PROGRAM Jog_Axis
VAR
	fbJog: MC_Jog;
	JogForwardPB: BOOL;
	JogBackwardsPB: BOOL;
END_VAR

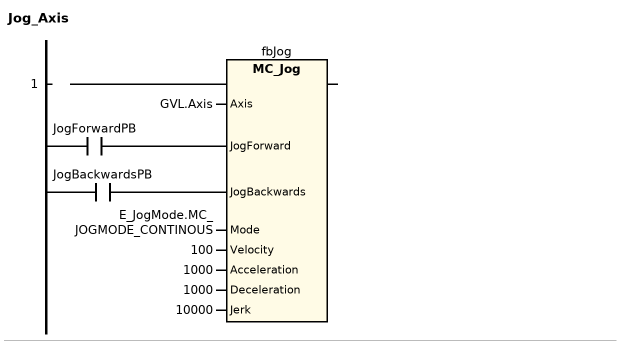
// NETWORK 1
fbJog(
    Axis := GVL.Axis,
    JogForward := JogForwardPB,
    JogBackwards := JogBackwardsPB,
    Mode := E_JogMode.MC_JOGMODE_CONTINOUS,
    Velocity := 100,
    Acceleration := 1000,
    Deceleration := 1000,
    Jerk := 10000); // MC_Jog

END_PROGRAM

(* stored: Version 1.1.0.1, ProductVersion 3.1.4024.12
   POU Jog_Axis: Id {cc0138ec-a5ac-423f-945f-45835e6f6566}, SpecialFunc None *)
